Xinje XDPPro project, PLC1: XD5-48T6 (software 3.5.3 2018-11-19)

PROGRAM Ladder

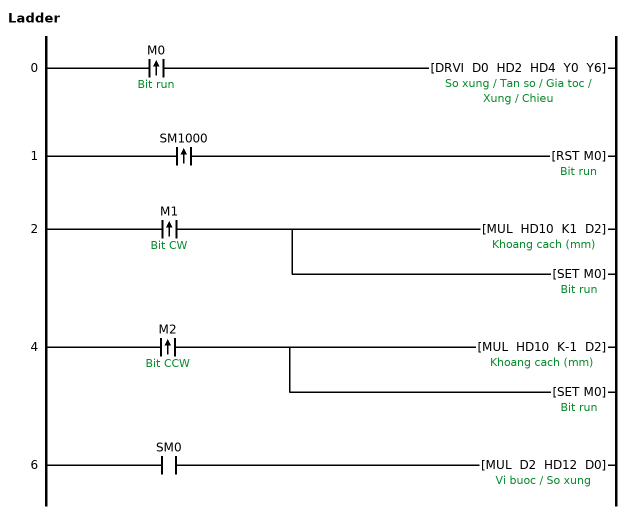
LDP    M0	; Bit run
DRVI   D0 HD2 HD4 Y0 Y6	; So xung / Tan so / Gia toc / Xung / Chieu
LDP    SM1000
RST    M0	; Bit run
LDP    M1	; Bit CW
MUL    HD10 K1 D2	; Khoang cach (mm)
SET    M0	; Bit run
LDP    M2	; Bit CCW
MUL    HD10 K-1 D2	; Khoang cach (mm)
SET    M0	; Bit run
LD     SM0
MUL    D2 HD12 D0	; Vi buoc / So xung